REGION Network 97: CLOSED LOW PRESSURE OUTPUT COMMAND MISSING ALARM
   RUNG wire#powerrail
      Contact( #M_VERIFY_LOW_PRESSURE )
      I_Contact( #CYL.CLOSE_LOW_PRESSURE )
      Contact( #CHECK_CLOSED_LOW_PRESSURE_CNC_PLC_SIGNAL )
      wire#w1
      Contact( #O_BYTE_0.CLOSED_LOW_PRESSURE_INPUT )
      Coil( #ALARMS.CLOSED_LOW_PRESSURE_OUTPUT_COMMAND_MISSING_ALARM )
   END_RUNG
   RUNG wire#powerrail
      Contact( #ALARMS.CLOSED_LOW_PRESSURE_OUTPUT_COMMAND_MISSING_ALARM )
      I_Contact( "DB2120_MPP_ITC_IPC".RESET_FAULTS )
   END_RUNG wire#w1
   // the same network as SCL:
   #ALARMS.CLOSED_LOW_PRESSURE_OUTPUT_COMMAND_MISSING_ALARM := ((#M_VERIFY_LOW_PRESSURE AND NOT #CYL.CLOSE_LOW_PRESSURE AND #CHECK_CLOSED_LOW_PRESSURE_CNC_PLC_SIGNAL) OR (#ALARMS.CLOSED_LOW_PRESSURE_OUTPUT_COMMAND_MISSING_ALARM AND NOT "DB2120_MPP_ITC_IPC".RESET_FAULTS)) AND #O_BYTE_0.CLOSED_LOW_PRESSURE_INPUT;
END_REGION

REGION Network 98: OPEN LOW PRESSURE TIME EXCEEDED ALARM
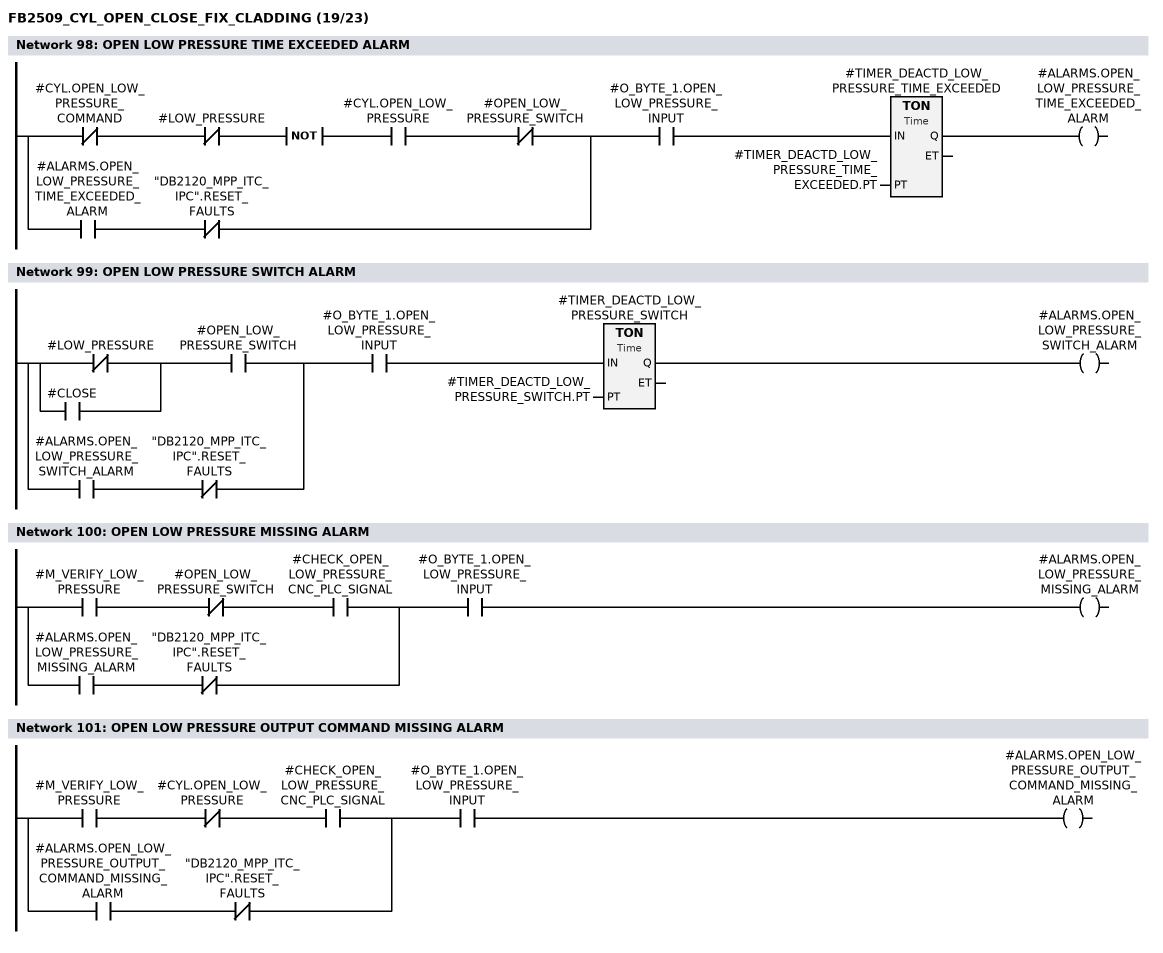
   RUNG wire#powerrail
      I_Contact( #CYL.OPEN_LOW_PRESSURE_COMMAND )
      I_Contact( #LOW_PRESSURE )
      Not()
      Contact( #CYL.OPEN_LOW_PRESSURE )
      I_Contact( #OPEN_LOW_PRESSURE_SWITCH )
      wire#w1
      Contact( #O_BYTE_1.OPEN_LOW_PRESSURE_INPUT )
      { S7_Templates := "time_type := Time" } #TIMER_DEACTD_LOW_PRESSURE_TIME_EXCEEDED.TON(pt := #TIMER_DEACTD_LOW_PRESSURE_TIME_EXCEEDED.PT, et =>)
      Coil( #ALARMS.OPEN_LOW_PRESSURE_TIME_EXCEEDED_ALARM )
   END_RUNG
   RUNG wire#powerrail
      Contact( #ALARMS.OPEN_LOW_PRESSURE_TIME_EXCEEDED_ALARM )
      I_Contact( "DB2120_MPP_ITC_IPC".RESET_FAULTS )
   END_RUNG wire#w1
   // the same network as SCL:
   #TIMER_DEACTD_LOW_PRESSURE_TIME_EXCEEDED(IN := ((NOT (NOT #CYL.OPEN_LOW_PRESSURE_COMMAND AND NOT #LOW_PRESSURE) AND #CYL.OPEN_LOW_PRESSURE AND NOT #OPEN_LOW_PRESSURE_SWITCH) OR (#ALARMS.OPEN_LOW_PRESSURE_TIME_EXCEEDED_ALARM AND NOT "DB2120_MPP_ITC_IPC".RESET_FAULTS)) AND #O_BYTE_1.OPEN_LOW_PRESSURE_INPUT,   // TON
                           PT := #TIMER_DEACTD_LOW_PRESSURE_TIME_EXCEEDED.PT);
   #ALARMS.OPEN_LOW_PRESSURE_TIME_EXCEEDED_ALARM := #TIMER_DEACTD_LOW_PRESSURE_TIME_EXCEEDED.Q;
END_REGION

REGION Network 99: OPEN LOW PRESSURE SWITCH ALARM
   RUNG wire#powerrail
      I_Contact( #LOW_PRESSURE )
      wire#w1
      Contact( #OPEN_LOW_PRESSURE_SWITCH )
      wire#w2
      Contact( #O_BYTE_1.OPEN_LOW_PRESSURE_INPUT )
      { S7_Templates := "time_type := Time" } #TIMER_DEACTD_LOW_PRESSURE_SWITCH.TON(pt := #TIMER_DEACTD_LOW_PRESSURE_SWITCH.PT, et =>)
      Coil( #ALARMS.OPEN_LOW_PRESSURE_SWITCH_ALARM )
   END_RUNG
   RUNG wire#powerrail
      Contact( #CLOSE )
   END_RUNG wire#w1
   RUNG wire#powerrail
      Contact( #ALARMS.OPEN_LOW_PRESSURE_SWITCH_ALARM )
      I_Contact( "DB2120_MPP_ITC_IPC".RESET_FAULTS )
   END_RUNG wire#w2
   // the same network as SCL:
   #TIMER_DEACTD_LOW_PRESSURE_SWITCH(IN := (((NOT #LOW_PRESSURE OR #CLOSE) AND #OPEN_LOW_PRESSURE_SWITCH) OR (#ALARMS.OPEN_LOW_PRESSURE_SWITCH_ALARM AND NOT "DB2120_MPP_ITC_IPC".RESET_FAULTS)) AND #O_BYTE_1.OPEN_LOW_PRESSURE_INPUT,   // TON
                           PT := #TIMER_DEACTD_LOW_PRESSURE_SWITCH.PT);
   #ALARMS.OPEN_LOW_PRESSURE_SWITCH_ALARM := #TIMER_DEACTD_LOW_PRESSURE_SWITCH.Q;
END_REGION

REGION Network 100: OPEN LOW PRESSURE MISSING ALARM
   RUNG wire#powerrail
      Contact( #M_VERIFY_LOW_PRESSURE )
      I_Contact( #OPEN_LOW_PRESSURE_SWITCH )
      Contact( #CHECK_OPEN_LOW_PRESSURE_CNC_PLC_SIGNAL )
      wire#w1
      Contact( #O_BYTE_1.OPEN_LOW_PRESSURE_INPUT )
      Coil( #ALARMS.OPEN_LOW_PRESSURE_MISSING_ALARM )
   END_RUNG
   RUNG wire#powerrail
      Contact( #ALARMS.OPEN_LOW_PRESSURE_MISSING_ALARM )
      I_Contact( "DB2120_MPP_ITC_IPC".RESET_FAULTS )
   END_RUNG wire#w1
   // the same network as SCL:
   #ALARMS.OPEN_LOW_PRESSURE_MISSING_ALARM := ((#M_VERIFY_LOW_PRESSURE AND NOT #OPEN_LOW_PRESSURE_SWITCH AND #CHECK_OPEN_LOW_PRESSURE_CNC_PLC_SIGNAL) OR (#ALARMS.OPEN_LOW_PRESSURE_MISSING_ALARM AND NOT "DB2120_MPP_ITC_IPC".RESET_FAULTS)) AND #O_BYTE_1.OPEN_LOW_PRESSURE_INPUT;
END_REGION

REGION Network 101: OPEN LOW PRESSURE OUTPUT COMMAND MISSING ALARM
   RUNG wire#powerrail
      Contact( #M_VERIFY_LOW_PRESSURE )
      I_Contact( #CYL.OPEN_LOW_PRESSURE )
      Contact( #CHECK_OPEN_LOW_PRESSURE_CNC_PLC_SIGNAL )
      wire#w1
      Contact( #O_BYTE_1.OPEN_LOW_PRESSURE_INPUT )
      Coil( #ALARMS.OPEN_LOW_PRESSURE_OUTPUT_COMMAND_MISSING_ALARM )
   END_RUNG
   RUNG wire#powerrail
      Contact( #ALARMS.OPEN_LOW_PRESSURE_OUTPUT_COMMAND_MISSING_ALARM )
      I_Contact( "DB2120_MPP_ITC_IPC".RESET_FAULTS )
   END_RUNG wire#w1
   // the same network as SCL:
   #ALARMS.OPEN_LOW_PRESSURE_OUTPUT_COMMAND_MISSING_ALARM := ((#M_VERIFY_LOW_PRESSURE AND NOT #CYL.OPEN_LOW_PRESSURE AND #CHECK_OPEN_LOW_PRESSURE_CNC_PLC_SIGNAL) OR (#ALARMS.OPEN_LOW_PRESSURE_OUTPUT_COMMAND_MISSING_ALARM AND NOT "DB2120_MPP_ITC_IPC".RESET_FAULTS)) AND #O_BYTE_1.OPEN_LOW_PRESSURE_INPUT;
END_REGION

REGION Network 102: RETURN HOME POSITION AND STOP END OF CYCLE ALARMS
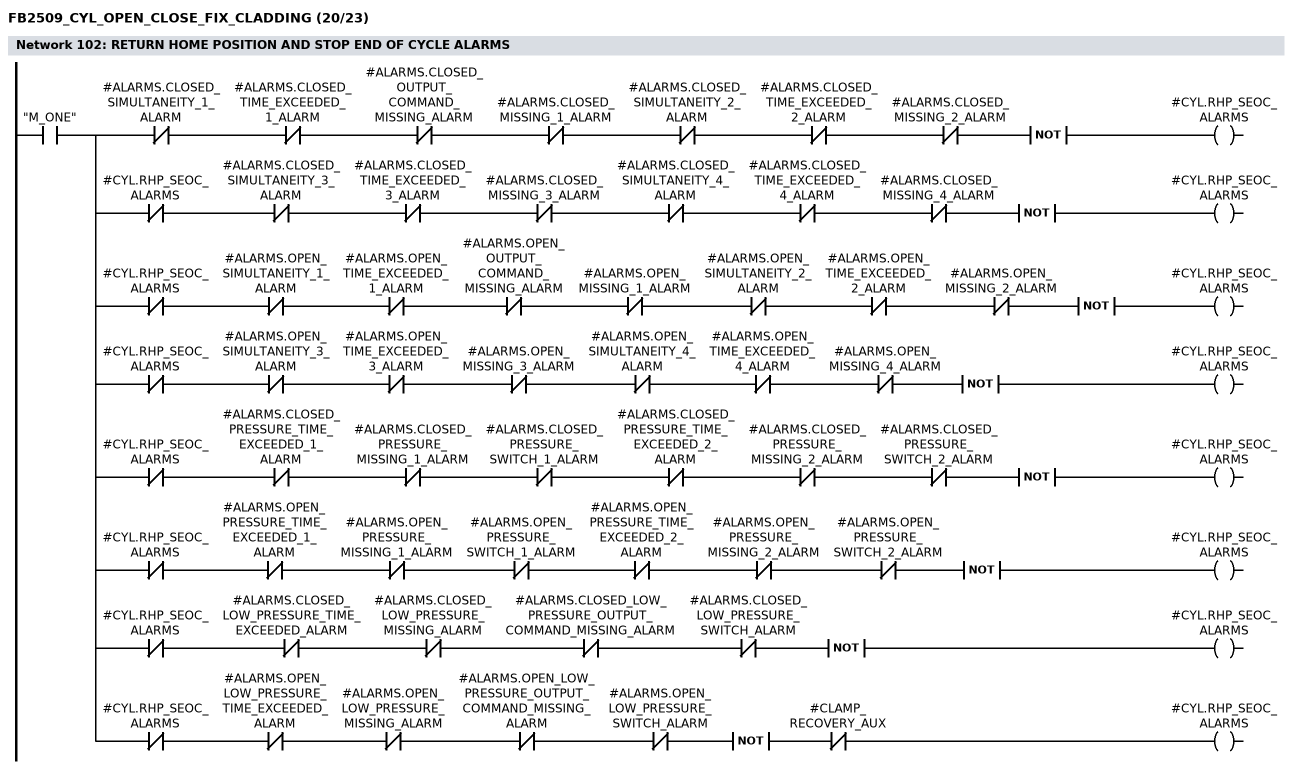
   RUNG wire#powerrail
      Contact( "M_ONE" )
      wire#w1
      I_Contact( #ALARMS.CLOSED_SIMULTANEITY_1_ALARM )
      I_Contact( #ALARMS.CLOSED_TIME_EXCEEDED_1_ALARM )
      I_Contact( #ALARMS.CLOSED_OUTPUT_COMMAND_MISSING_ALARM )
      I_Contact( #ALARMS.CLOSED_MISSING_1_ALARM )
      I_Contact( #ALARMS.CLOSED_SIMULTANEITY_2_ALARM )
      I_Contact( #ALARMS.CLOSED_TIME_EXCEEDED_2_ALARM )
      I_Contact( #ALARMS.CLOSED_MISSING_2_ALARM )
      Not()
      Coil( #CYL.RHP_SEOC_ALARMS )
   END_RUNG
   RUNG wire#w1
      I_Contact( #CYL.RHP_SEOC_ALARMS )
      I_Contact( #ALARMS.CLOSED_SIMULTANEITY_3_ALARM )
      I_Contact( #ALARMS.CLOSED_TIME_EXCEEDED_3_ALARM )
      I_Contact( #ALARMS.CLOSED_MISSING_3_ALARM )
      I_Contact( #ALARMS.CLOSED_SIMULTANEITY_4_ALARM )
      I_Contact( #ALARMS.CLOSED_TIME_EXCEEDED_4_ALARM )
      I_Contact( #ALARMS.CLOSED_MISSING_4_ALARM )
      Not()
      Coil( #CYL.RHP_SEOC_ALARMS )
   END_RUNG
   RUNG wire#w1
      I_Contact( #CYL.RHP_SEOC_ALARMS )
      I_Contact( #ALARMS.OPEN_SIMULTANEITY_1_ALARM )
      I_Contact( #ALARMS.OPEN_TIME_EXCEEDED_1_ALARM )
      I_Contact( #ALARMS.OPEN_OUTPUT_COMMAND_MISSING_ALARM )
      I_Contact( #ALARMS.OPEN_MISSING_1_ALARM )
      I_Contact( #ALARMS.OPEN_SIMULTANEITY_2_ALARM )
      I_Contact( #ALARMS.OPEN_TIME_EXCEEDED_2_ALARM )
      I_Contact( #ALARMS.OPEN_MISSING_2_ALARM )
      Not()
      Coil( #CYL.RHP_SEOC_ALARMS )
   END_RUNG
   RUNG wire#w1
      I_Contact( #CYL.RHP_SEOC_ALARMS )
      I_Contact( #ALARMS.OPEN_SIMULTANEITY_3_ALARM )
      I_Contact( #ALARMS.OPEN_TIME_EXCEEDED_3_ALARM )
      I_Contact( #ALARMS.OPEN_MISSING_3_ALARM )
      I_Contact( #ALARMS.OPEN_SIMULTANEITY_4_ALARM )
      I_Contact( #ALARMS.OPEN_TIME_EXCEEDED_4_ALARM )
      I_Contact( #ALARMS.OPEN_MISSING_4_ALARM )
      Not()
      Coil( #CYL.RHP_SEOC_ALARMS )
   END_RUNG
   RUNG wire#w1
      I_Contact( #CYL.RHP_SEOC_ALARMS )
      I_Contact( #ALARMS.CLOSED_PRESSURE_TIME_EXCEEDED_1_ALARM )
      I_Contact( #ALARMS.CLOSED_PRESSURE_MISSING_1_ALARM )
      I_Contact( #ALARMS.CLOSED_PRESSURE_SWITCH_1_ALARM )
      I_Contact( #ALARMS.CLOSED_PRESSURE_TIME_EXCEEDED_2_ALARM )
      I_Contact( #ALARMS.CLOSED_PRESSURE_MISSING_2_ALARM )
      I_Contact( #ALARMS.CLOSED_PRESSURE_SWITCH_2_ALARM )
      Not()
      Coil( #CYL.RHP_SEOC_ALARMS )
   END_RUNG
   RUNG wire#w1
      I_Contact( #CYL.RHP_SEOC_ALARMS )
      I_Contact( #ALARMS.OPEN_PRESSURE_TIME_EXCEEDED_1_ALARM )
      I_Contact( #ALARMS.OPEN_PRESSURE_MISSING_1_ALARM )
      I_Contact( #ALARMS.OPEN_PRESSURE_SWITCH_1_ALARM )
      I_Contact( #ALARMS.OPEN_PRESSURE_TIME_EXCEEDED_2_ALARM )
      I_Contact( #ALARMS.OPEN_PRESSURE_MISSING_2_ALARM )
      I_Contact( #ALARMS.OPEN_PRESSURE_SWITCH_2_ALARM )
      Not()
      Coil( #CYL.RHP_SEOC_ALARMS )
   END_RUNG
   RUNG wire#w1
      I_Contact( #CYL.RHP_SEOC_ALARMS )
      I_Contact( #ALARMS.CLOSED_LOW_PRESSURE_TIME_EXCEEDED_ALARM )
      I_Contact( #ALARMS.CLOSED_LOW_PRESSURE_MISSING_ALARM )
      I_Contact( #ALARMS.CLOSED_LOW_PRESSURE_OUTPUT_COMMAND_MISSING_ALARM )
      I_Contact( #ALARMS.CLOSED_LOW_PRESSURE_SWITCH_ALARM )
      Not()
      Coil( #CYL.RHP_SEOC_ALARMS )
   END_RUNG
   RUNG wire#w1
      I_Contact( #CYL.RHP_SEOC_ALARMS )
      I_Contact( #ALARMS.OPEN_LOW_PRESSURE_TIME_EXCEEDED_ALARM )
      I_Contact( #ALARMS.OPEN_LOW_PRESSURE_MISSING_ALARM )
      I_Contact( #ALARMS.OPEN_LOW_PRESSURE_OUTPUT_COMMAND_MISSING_ALARM )
      I_Contact( #ALARMS.OPEN_LOW_PRESSURE_SWITCH_ALARM )
      Not()
      I_Contact( #CLAMP_RECOVERY_AUX )
      Coil( #CYL.RHP_SEOC_ALARMS )
   END_RUNG
   // the same network as SCL:
   #CYL.RHP_SEOC_ALARMS := NOT ("M_ONE" AND NOT #ALARMS.CLOSED_SIMULTANEITY_1_ALARM AND NOT #ALARMS.CLOSED_TIME_EXCEEDED_1_ALARM AND NOT #ALARMS.CLOSED_OUTPUT_COMMAND_MISSING_ALARM AND NOT #ALARMS.CLOSED_MISSING_1_ALARM AND NOT #ALARMS.CLOSED_SIMULTANEITY_2_ALARM AND NOT #ALARMS.CLOSED_TIME_EXCEEDED_2_ALARM AND NOT #ALARMS.CLOSED_MISSING_2_ALARM);
   #CYL.RHP_SEOC_ALARMS := NOT ("M_ONE" AND NOT #CYL.RHP_SEOC_ALARMS AND NOT #ALARMS.CLOSED_SIMULTANEITY_3_ALARM AND NOT #ALARMS.CLOSED_TIME_EXCEEDED_3_ALARM AND NOT #ALARMS.CLOSED_MISSING_3_ALARM AND NOT #ALARMS.CLOSED_SIMULTANEITY_4_ALARM AND NOT #ALARMS.CLOSED_TIME_EXCEEDED_4_ALARM AND NOT #ALARMS.CLOSED_MISSING_4_ALARM);
   #CYL.RHP_SEOC_ALARMS := NOT ("M_ONE" AND NOT #CYL.RHP_SEOC_ALARMS AND NOT #ALARMS.OPEN_SIMULTANEITY_1_ALARM AND NOT #ALARMS.OPEN_TIME_EXCEEDED_1_ALARM AND NOT #ALARMS.OPEN_OUTPUT_COMMAND_MISSING_ALARM AND NOT #ALARMS.OPEN_MISSING_1_ALARM AND NOT #ALARMS.OPEN_SIMULTANEITY_2_ALARM AND NOT #ALARMS.OPEN_TIME_EXCEEDED_2_ALARM AND NOT #ALARMS.OPEN_MISSING_2_ALARM);
   #CYL.RHP_SEOC_ALARMS := NOT ("M_ONE" AND NOT #CYL.RHP_SEOC_ALARMS AND NOT #ALARMS.OPEN_SIMULTANEITY_3_ALARM AND NOT #ALARMS.OPEN_TIME_EXCEEDED_3_ALARM AND NOT #ALARMS.OPEN_MISSING_3_ALARM AND NOT #ALARMS.OPEN_SIMULTANEITY_4_ALARM AND NOT #ALARMS.OPEN_TIME_EXCEEDED_4_ALARM AND NOT #ALARMS.OPEN_MISSING_4_ALARM);
   #CYL.RHP_SEOC_ALARMS := NOT ("M_ONE" AND NOT #CYL.RHP_SEOC_ALARMS AND NOT #ALARMS.CLOSED_PRESSURE_TIME_EXCEEDED_1_ALARM AND NOT #ALARMS.CLOSED_PRESSURE_MISSING_1_ALARM AND NOT #ALARMS.CLOSED_PRESSURE_SWITCH_1_ALARM AND NOT #ALARMS.CLOSED_PRESSURE_TIME_EXCEEDED_2_ALARM AND NOT #ALARMS.CLOSED_PRESSURE_MISSING_2_ALARM AND NOT #ALARMS.CLOSED_PRESSURE_SWITCH_2_ALARM);
   #CYL.RHP_SEOC_ALARMS := NOT ("M_ONE" AND NOT #CYL.RHP_SEOC_ALARMS AND NOT #ALARMS.OPEN_PRESSURE_TIME_EXCEEDED_1_ALARM AND NOT #ALARMS.OPEN_PRESSURE_MISSING_1_ALARM AND NOT #ALARMS.OPEN_PRESSURE_SWITCH_1_ALARM AND NOT #ALARMS.OPEN_PRESSURE_TIME_EXCEEDED_2_ALARM AND NOT #ALARMS.OPEN_PRESSURE_MISSING_2_ALARM AND NOT #ALARMS.OPEN_PRESSURE_SWITCH_2_ALARM);
   #CYL.RHP_SEOC_ALARMS := NOT ("M_ONE" AND NOT #CYL.RHP_SEOC_ALARMS AND NOT #ALARMS.CLOSED_LOW_PRESSURE_TIME_EXCEEDED_ALARM AND NOT #ALARMS.CLOSED_LOW_PRESSURE_MISSING_ALARM AND NOT #ALARMS.CLOSED_LOW_PRESSURE_OUTPUT_COMMAND_MISSING_ALARM AND NOT #ALARMS.CLOSED_LOW_PRESSURE_SWITCH_ALARM);
   #CYL.RHP_SEOC_ALARMS := NOT ("M_ONE" AND NOT #CYL.RHP_SEOC_ALARMS AND NOT #ALARMS.OPEN_LOW_PRESSURE_TIME_EXCEEDED_ALARM AND NOT #ALARMS.OPEN_LOW_PRESSURE_MISSING_ALARM AND NOT #ALARMS.OPEN_LOW_PRESSURE_OUTPUT_COMMAND_MISSING_ALARM AND NOT #ALARMS.OPEN_LOW_PRESSURE_SWITCH_ALARM) AND NOT #CLAMP_RECOVERY_AUX;
END_REGION

REGION Network 103: RETURN HOME POSITION AND STOP END OF CYCLE ALARMS
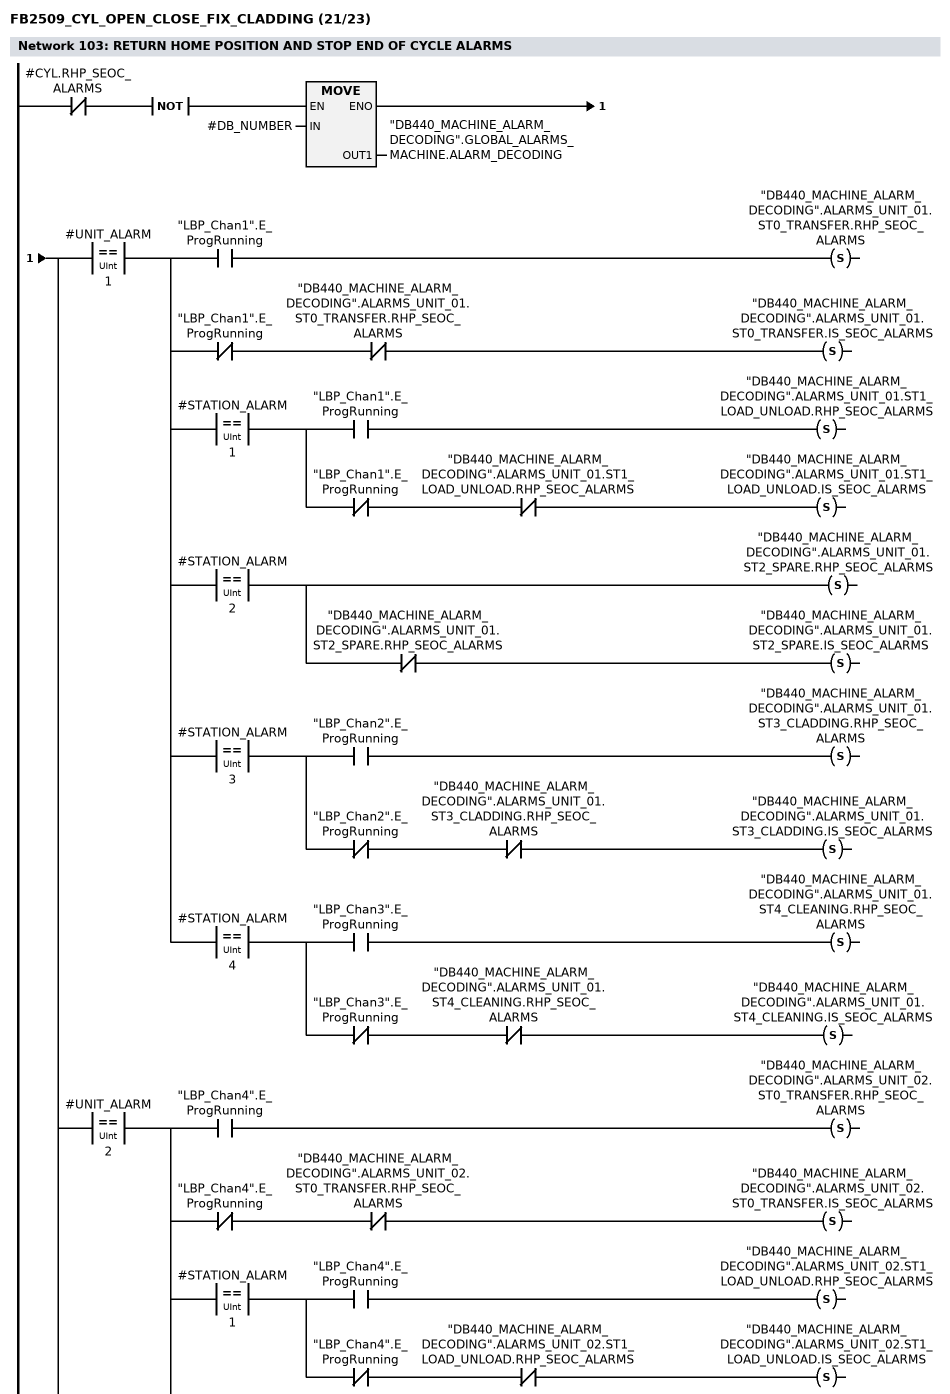
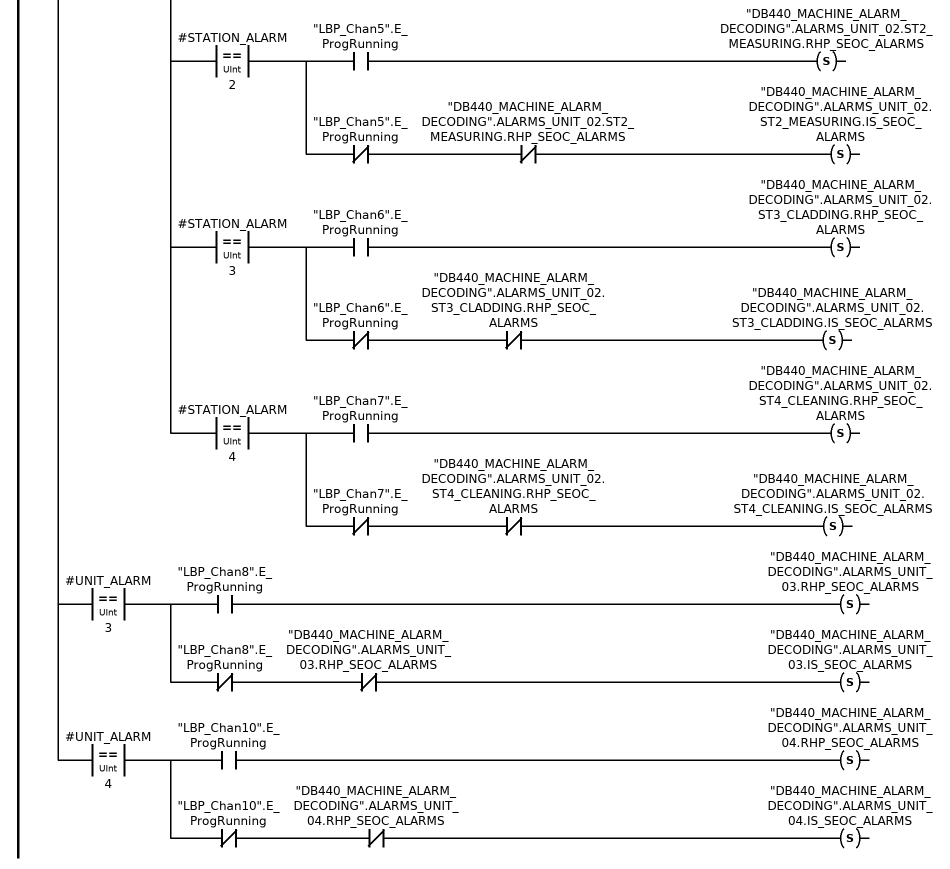
   RUNG wire#powerrail
      I_Contact( #CYL.RHP_SEOC_ALARMS )
      Not()
      { S7_GenerateENO := "TRUE" } Move(in := #DB_NUMBER, out1 => "DB440_MACHINE_ALARM_DECODING".GLOBAL_ALARMS_MACHINE.ALARM_DECODING)
      wire#w1
      { S7_Templates := "SrcType := UInt" } EQ_Contact(in1 := #UNIT_ALARM, in2 := 1)
      wire#w2
      Contact( "LBP_Chan1".E_ProgRunning )
      S_Coil( "DB440_MACHINE_ALARM_DECODING".ALARMS_UNIT_01.ST0_TRANSFER.RHP_SEOC_ALARMS )
   END_RUNG
   RUNG wire#w2
      I_Contact( "LBP_Chan1".E_ProgRunning )
      I_Contact( "DB440_MACHINE_ALARM_DECODING".ALARMS_UNIT_01.ST0_TRANSFER.RHP_SEOC_ALARMS )
      S_Coil( "DB440_MACHINE_ALARM_DECODING".ALARMS_UNIT_01.ST0_TRANSFER.IS_SEOC_ALARMS )
   END_RUNG
   RUNG wire#w2
      { S7_Templates := "SrcType := UInt" } EQ_Contact(in1 := #STATION_ALARM, in2 := 1)
      wire#w3
      Contact( "LBP_Chan1".E_ProgRunning )
      S_Coil( "DB440_MACHINE_ALARM_DECODING".ALARMS_UNIT_01.ST1_LOAD_UNLOAD.RHP_SEOC_ALARMS )
   END_RUNG
   RUNG wire#w3
      I_Contact( "LBP_Chan1".E_ProgRunning )
      I_Contact( "DB440_MACHINE_ALARM_DECODING".ALARMS_UNIT_01.ST1_LOAD_UNLOAD.RHP_SEOC_ALARMS )
      S_Coil( "DB440_MACHINE_ALARM_DECODING".ALARMS_UNIT_01.ST1_LOAD_UNLOAD.IS_SEOC_ALARMS )
   END_RUNG
   RUNG wire#w2
      { S7_Templates := "SrcType := UInt" } EQ_Contact(in1 := #STATION_ALARM, in2 := 2)
      wire#w4
      S_Coil( "DB440_MACHINE_ALARM_DECODING".ALARMS_UNIT_01.ST2_SPARE.RHP_SEOC_ALARMS )
   END_RUNG
   RUNG wire#w4
      I_Contact( "DB440_MACHINE_ALARM_DECODING".ALARMS_UNIT_01.ST2_SPARE.RHP_SEOC_ALARMS )
      S_Coil( "DB440_MACHINE_ALARM_DECODING".ALARMS_UNIT_01.ST2_SPARE.IS_SEOC_ALARMS )
   END_RUNG
   RUNG wire#w2
      { S7_Templates := "SrcType := UInt" } EQ_Contact(in1 := #STATION_ALARM, in2 := 3)
      wire#w5
      Contact( "LBP_Chan2".E_ProgRunning )
      S_Coil( "DB440_MACHINE_ALARM_DECODING".ALARMS_UNIT_01.ST3_CLADDING.RHP_SEOC_ALARMS )
   END_RUNG
   RUNG wire#w5
      I_Contact( "LBP_Chan2".E_ProgRunning )
      I_Contact( "DB440_MACHINE_ALARM_DECODING".ALARMS_UNIT_01.ST3_CLADDING.RHP_SEOC_ALARMS )
      S_Coil( "DB440_MACHINE_ALARM_DECODING".ALARMS_UNIT_01.ST3_CLADDING.IS_SEOC_ALARMS )
   END_RUNG
   RUNG wire#w2
      { S7_Templates := "SrcType := UInt" } EQ_Contact(in1 := #STATION_ALARM, in2 := 4)
      wire#w6
      Contact( "LBP_Chan3".E_ProgRunning )
      S_Coil( "DB440_MACHINE_ALARM_DECODING".ALARMS_UNIT_01.ST4_CLEANING.RHP_SEOC_ALARMS )
   END_RUNG
   RUNG wire#w6
      I_Contact( "LBP_Chan3".E_ProgRunning )
      I_Contact( "DB440_MACHINE_ALARM_DECODING".ALARMS_UNIT_01.ST4_CLEANING.RHP_SEOC_ALARMS )
      S_Coil( "DB440_MACHINE_ALARM_DECODING".ALARMS_UNIT_01.ST4_CLEANING.IS_SEOC_ALARMS )
   END_RUNG
   RUNG wire#w1
      { S7_Templates := "SrcType := UInt" } EQ_Contact(in1 := #UNIT_ALARM, in2 := 2)
      wire#w7
      Contact( "LBP_Chan4".E_ProgRunning )
      S_Coil( "DB440_MACHINE_ALARM_DECODING".ALARMS_UNIT_02.ST0_TRANSFER.RHP_SEOC_ALARMS )
   END_RUNG
   RUNG wire#w7
      I_Contact( "LBP_Chan4".E_ProgRunning )
      I_Contact( "DB440_MACHINE_ALARM_DECODING".ALARMS_UNIT_02.ST0_TRANSFER.RHP_SEOC_ALARMS )
      S_Coil( "DB440_MACHINE_ALARM_DECODING".ALARMS_UNIT_02.ST0_TRANSFER.IS_SEOC_ALARMS )
   END_RUNG
   RUNG wire#w7
      { S7_Templates := "SrcType := UInt" } EQ_Contact(in1 := #STATION_ALARM, in2 := 1)
      wire#w8
      Contact( "LBP_Chan4".E_ProgRunning )
      S_Coil( "DB440_MACHINE_ALARM_DECODING".ALARMS_UNIT_02.ST1_LOAD_UNLOAD.RHP_SEOC_ALARMS )
   END_RUNG
   RUNG wire#w8
      I_Contact( "LBP_Chan4".E_ProgRunning )
      I_Contact( "DB440_MACHINE_ALARM_DECODING".ALARMS_UNIT_02.ST1_LOAD_UNLOAD.RHP_SEOC_ALARMS )
      S_Coil( "DB440_MACHINE_ALARM_DECODING".ALARMS_UNIT_02.ST1_LOAD_UNLOAD.IS_SEOC_ALARMS )
   END_RUNG
   RUNG wire#w7
      { S7_Templates := "SrcType := UInt" } EQ_Contact(in1 := #STATION_ALARM, in2 := 2)
      wire#w9
      Contact( "LBP_Chan5".E_ProgRunning )
      S_Coil( "DB440_MACHINE_ALARM_DECODING".ALARMS_UNIT_02.ST2_MEASURING.RHP_SEOC_ALARMS )
   END_RUNG
   RUNG wire#w9
      I_Contact( "LBP_Chan5".E_ProgRunning )
      I_Contact( "DB440_MACHINE_ALARM_DECODING".ALARMS_UNIT_02.ST2_MEASURING.RHP_SEOC_ALARMS )
      S_Coil( "DB440_MACHINE_ALARM_DECODING".ALARMS_UNIT_02.ST2_MEASURING.IS_SEOC_ALARMS )
   END_RUNG
   RUNG wire#w7
      { S7_Templates := "SrcType := UInt" } EQ_Contact(in1 := #STATION_ALARM, in2 := 3)
      wire#w10
      Contact( "LBP_Chan6".E_ProgRunning )
      S_Coil( "DB440_MACHINE_ALARM_DECODING".ALARMS_UNIT_02.ST3_CLADDING.RHP_SEOC_ALARMS )
   END_RUNG
   RUNG wire#w10
      I_Contact( "LBP_Chan6".E_ProgRunning )
      I_Contact( "DB440_MACHINE_ALARM_DECODING".ALARMS_UNIT_02.ST3_CLADDING.RHP_SEOC_ALARMS )
      S_Coil( "DB440_MACHINE_ALARM_DECODING".ALARMS_UNIT_02.ST3_CLADDING.IS_SEOC_ALARMS )
   END_RUNG
   RUNG wire#w7
      { S7_Templates := "SrcType := UInt" } EQ_Contact(in1 := #STATION_ALARM, in2 := 4)
      wire#w11
      Contact( "LBP_Chan7".E_ProgRunning )
      S_Coil( "DB440_MACHINE_ALARM_DECODING".ALARMS_UNIT_02.ST4_CLEANING.RHP_SEOC_ALARMS )
   END_RUNG
   RUNG wire#w11
      I_Contact( "LBP_Chan7".E_ProgRunning )
      I_Contact( "DB440_MACHINE_ALARM_DECODING".ALARMS_UNIT_02.ST4_CLEANING.RHP_SEOC_ALARMS )
      S_Coil( "DB440_MACHINE_ALARM_DECODING".ALARMS_UNIT_02.ST4_CLEANING.IS_SEOC_ALARMS )
   END_RUNG
   RUNG wire#w1
      { S7_Templates := "SrcType := UInt" } EQ_Contact(in1 := #UNIT_ALARM, in2 := 3)
      wire#w12
      Contact( "LBP_Chan8".E_ProgRunning )
      S_Coil( "DB440_MACHINE_ALARM_DECODING".ALARMS_UNIT_03.RHP_SEOC_ALARMS )
   END_RUNG
   RUNG wire#w12
      I_Contact( "LBP_Chan8".E_ProgRunning )
      I_Contact( "DB440_MACHINE_ALARM_DECODING".ALARMS_UNIT_03.RHP_SEOC_ALARMS )
      S_Coil( "DB440_MACHINE_ALARM_DECODING".ALARMS_UNIT_03.IS_SEOC_ALARMS )
   END_RUNG
   RUNG wire#w1
      { S7_Templates := "SrcType := UInt" } EQ_Contact(in1 := #UNIT_ALARM, in2 := 4)
      wire#w13
      Contact( "LBP_Chan10".E_ProgRunning )
      S_Coil( "DB440_MACHINE_ALARM_DECODING".ALARMS_UNIT_04.RHP_SEOC_ALARMS )
   END_RUNG
   RUNG wire#w13
      I_Contact( "LBP_Chan10".E_ProgRunning )
      I_Contact( "DB440_MACHINE_ALARM_DECODING".ALARMS_UNIT_04.RHP_SEOC_ALARMS )
      S_Coil( "DB440_MACHINE_ALARM_DECODING".ALARMS_UNIT_04.IS_SEOC_ALARMS )
   END_RUNG
   // the same network as SCL:
   // ENO of a box is taken as its EN; it also drops when the box reports an error
   #_w1 := NOT (NOT #CYL.RHP_SEOC_ALARMS);
   IF #_w1 THEN "DB440_MACHINE_ALARM_DECODING".GLOBAL_ALARMS_MACHINE.ALARM_DECODING := #DB_NUMBER; END_IF;
   #_w2 := #_w1 AND (#UNIT_ALARM = 1);
   IF #_w2 AND "LBP_Chan1".E_ProgRunning THEN
       "DB440_MACHINE_ALARM_DECODING".ALARMS_UNIT_01.ST0_TRANSFER.RHP_SEOC_ALARMS := TRUE;
   END_IF;
   IF #_w2 AND NOT "LBP_Chan1".E_ProgRunning AND NOT "DB440_MACHINE_ALARM_DECODING".ALARMS_UNIT_01.ST0_TRANSFER.RHP_SEOC_ALARMS THEN
       "DB440_MACHINE_ALARM_DECODING".ALARMS_UNIT_01.ST0_TRANSFER.IS_SEOC_ALARMS := TRUE;
   END_IF;
   #_w3 := #_w2 AND (#STATION_ALARM = 1);
   IF #_w3 AND "LBP_Chan1".E_ProgRunning THEN
       "DB440_MACHINE_ALARM_DECODING".ALARMS_UNIT_01.ST1_LOAD_UNLOAD.RHP_SEOC_ALARMS := TRUE;
   END_IF;
   IF #_w3 AND NOT "LBP_Chan1".E_ProgRunning AND NOT "DB440_MACHINE_ALARM_DECODING".ALARMS_UNIT_01.ST1_LOAD_UNLOAD.RHP_SEOC_ALARMS THEN
       "DB440_MACHINE_ALARM_DECODING".ALARMS_UNIT_01.ST1_LOAD_UNLOAD.IS_SEOC_ALARMS := TRUE;
   END_IF;
   #_w4 := #_w2 AND (#STATION_ALARM = 2);
   IF #_w4 THEN "DB440_MACHINE_ALARM_DECODING".ALARMS_UNIT_01.ST2_SPARE.RHP_SEOC_ALARMS := TRUE; END_IF;
   IF #_w4 AND NOT "DB440_MACHINE_ALARM_DECODING".ALARMS_UNIT_01.ST2_SPARE.RHP_SEOC_ALARMS THEN
       "DB440_MACHINE_ALARM_DECODING".ALARMS_UNIT_01.ST2_SPARE.IS_SEOC_ALARMS := TRUE;
   END_IF;
   #_w5 := #_w2 AND (#STATION_ALARM = 3);
   IF #_w5 AND "LBP_Chan2".E_ProgRunning THEN
       "DB440_MACHINE_ALARM_DECODING".ALARMS_UNIT_01.ST3_CLADDING.RHP_SEOC_ALARMS := TRUE;
   END_IF;
   IF #_w5 AND NOT "LBP_Chan2".E_ProgRunning AND NOT "DB440_MACHINE_ALARM_DECODING".ALARMS_UNIT_01.ST3_CLADDING.RHP_SEOC_ALARMS THEN
       "DB440_MACHINE_ALARM_DECODING".ALARMS_UNIT_01.ST3_CLADDING.IS_SEOC_ALARMS := TRUE;
   END_IF;
   #_w6 := #_w2 AND (#STATION_ALARM = 4);
   IF #_w6 AND "LBP_Chan3".E_ProgRunning THEN
       "DB440_MACHINE_ALARM_DECODING".ALARMS_UNIT_01.ST4_CLEANING.RHP_SEOC_ALARMS := TRUE;
   END_IF;
   IF #_w6 AND NOT "LBP_Chan3".E_ProgRunning AND NOT "DB440_MACHINE_ALARM_DECODING".ALARMS_UNIT_01.ST4_CLEANING.RHP_SEOC_ALARMS THEN
       "DB440_MACHINE_ALARM_DECODING".ALARMS_UNIT_01.ST4_CLEANING.IS_SEOC_ALARMS := TRUE;
   END_IF;
   #_w7 := #_w1 AND (#UNIT_ALARM = 2);
   IF #_w7 AND "LBP_Chan4".E_ProgRunning THEN
       "DB440_MACHINE_ALARM_DECODING".ALARMS_UNIT_02.ST0_TRANSFER.RHP_SEOC_ALARMS := TRUE;
   END_IF;
   IF #_w7 AND NOT "LBP_Chan4".E_ProgRunning AND NOT "DB440_MACHINE_ALARM_DECODING".ALARMS_UNIT_02.ST0_TRANSFER.RHP_SEOC_ALARMS THEN
       "DB440_MACHINE_ALARM_DECODING".ALARMS_UNIT_02.ST0_TRANSFER.IS_SEOC_ALARMS := TRUE;
   END_IF;
   #_w8 := #_w7 AND (#STATION_ALARM = 1);
   IF #_w8 AND "LBP_Chan4".E_ProgRunning THEN
       "DB440_MACHINE_ALARM_DECODING".ALARMS_UNIT_02.ST1_LOAD_UNLOAD.RHP_SEOC_ALARMS := TRUE;
   END_IF;
   IF #_w8 AND NOT "LBP_Chan4".E_ProgRunning AND NOT "DB440_MACHINE_ALARM_DECODING".ALARMS_UNIT_02.ST1_LOAD_UNLOAD.RHP_SEOC_ALARMS THEN
       "DB440_MACHINE_ALARM_DECODING".ALARMS_UNIT_02.ST1_LOAD_UNLOAD.IS_SEOC_ALARMS := TRUE;
   END_IF;
   #_w9 := #_w7 AND (#STATION_ALARM = 2);
   IF #_w9 AND "LBP_Chan5".E_ProgRunning THEN
       "DB440_MACHINE_ALARM_DECODING".ALARMS_UNIT_02.ST2_MEASURING.RHP_SEOC_ALARMS := TRUE;
   END_IF;
   IF #_w9 AND NOT "LBP_Chan5".E_ProgRunning AND NOT "DB440_MACHINE_ALARM_DECODING".ALARMS_UNIT_02.ST2_MEASURING.RHP_SEOC_ALARMS THEN
       "DB440_MACHINE_ALARM_DECODING".ALARMS_UNIT_02.ST2_MEASURING.IS_SEOC_ALARMS := TRUE;
   END_IF;
   #_w10 := #_w7 AND (#STATION_ALARM = 3);
   IF #_w10 AND "LBP_Chan6".E_ProgRunning THEN
       "DB440_MACHINE_ALARM_DECODING".ALARMS_UNIT_02.ST3_CLADDING.RHP_SEOC_ALARMS := TRUE;
   END_IF;
   IF #_w10 AND NOT "LBP_Chan6".E_ProgRunning AND NOT "DB440_MACHINE_ALARM_DECODING".ALARMS_UNIT_02.ST3_CLADDING.RHP_SEOC_ALARMS THEN
       "DB440_MACHINE_ALARM_DECODING".ALARMS_UNIT_02.ST3_CLADDING.IS_SEOC_ALARMS := TRUE;
   END_IF;
   #_w11 := #_w7 AND (#STATION_ALARM = 4);
   IF #_w11 AND "LBP_Chan7".E_ProgRunning THEN
       "DB440_MACHINE_ALARM_DECODING".ALARMS_UNIT_02.ST4_CLEANING.RHP_SEOC_ALARMS := TRUE;
   END_IF;
   IF #_w11 AND NOT "LBP_Chan7".E_ProgRunning AND NOT "DB440_MACHINE_ALARM_DECODING".ALARMS_UNIT_02.ST4_CLEANING.RHP_SEOC_ALARMS THEN
       "DB440_MACHINE_ALARM_DECODING".ALARMS_UNIT_02.ST4_CLEANING.IS_SEOC_ALARMS := TRUE;
   END_IF;
   #_w12 := #_w1 AND (#UNIT_ALARM = 3);
   IF #_w12 AND "LBP_Chan8".E_ProgRunning THEN
       "DB440_MACHINE_ALARM_DECODING".ALARMS_UNIT_03.RHP_SEOC_ALARMS := TRUE;
   END_IF;
   IF #_w12 AND NOT "LBP_Chan8".E_ProgRunning AND NOT "DB440_MACHINE_ALARM_DECODING".ALARMS_UNIT_03.RHP_SEOC_ALARMS THEN
       "DB440_MACHINE_ALARM_DECODING".ALARMS_UNIT_03.IS_SEOC_ALARMS := TRUE;
   END_IF;
   #_w13 := #_w1 AND (#UNIT_ALARM = 4);
   IF #_w13 AND "LBP_Chan10".E_ProgRunning THEN
       "DB440_MACHINE_ALARM_DECODING".ALARMS_UNIT_04.RHP_SEOC_ALARMS := TRUE;
   END_IF;
   IF #_w13 AND NOT "LBP_Chan10".E_ProgRunning AND NOT "DB440_MACHINE_ALARM_DECODING".ALARMS_UNIT_04.RHP_SEOC_ALARMS THEN
       "DB440_MACHINE_ALARM_DECODING".ALARMS_UNIT_04.IS_SEOC_ALARMS := TRUE;
   END_IF;
END_REGION

REGION Network 104: ANY ACTIVE ALARM
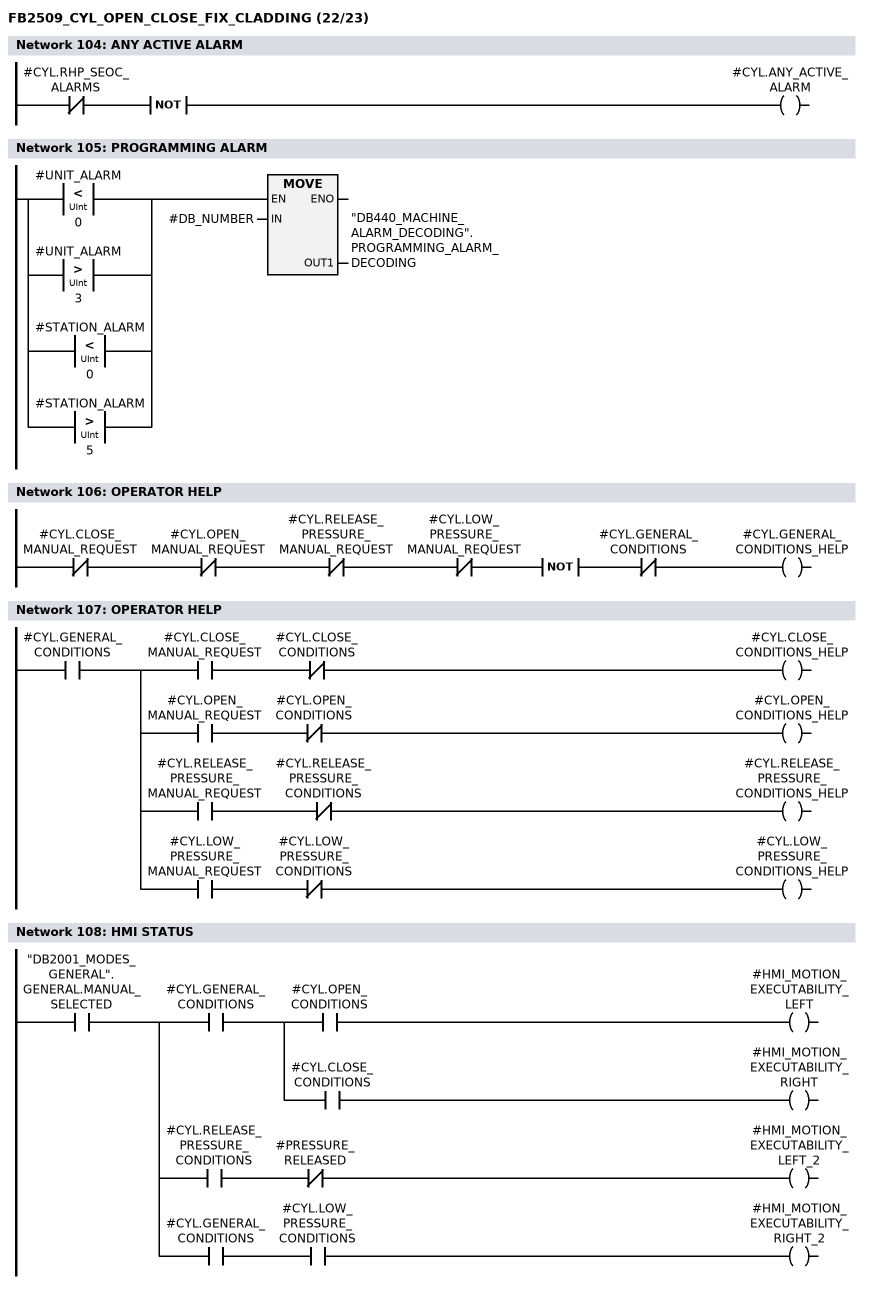
   RUNG wire#powerrail
      I_Contact( #CYL.RHP_SEOC_ALARMS )
      Not()
      Coil( #CYL.ANY_ACTIVE_ALARM )
   END_RUNG
   // the same network as SCL:
   #CYL.ANY_ACTIVE_ALARM := NOT (NOT #CYL.RHP_SEOC_ALARMS);
END_REGION

REGION Network 105: PROGRAMMING ALARM
   RUNG wire#powerrail
      { S7_Templates := "SrcType := UInt" } LT_Contact(in1 := #UNIT_ALARM, in2 := 0)
      wire#w1
      Move(in := #DB_NUMBER, out1 => "DB440_MACHINE_ALARM_DECODING".PROGRAMMING_ALARM_DECODING)
   END_RUNG
   RUNG wire#powerrail
      { S7_Templates := "SrcType := UInt" } GT_Contact(in1 := #UNIT_ALARM, in2 := 3)
   END_RUNG wire#w1
   RUNG wire#powerrail
      { S7_Templates := "SrcType := UInt" } LT_Contact(in1 := #STATION_ALARM, in2 := 0)
   END_RUNG wire#w1
   RUNG wire#powerrail
      { S7_Templates := "SrcType := UInt" } GT_Contact(in1 := #STATION_ALARM, in2 := 5)
   END_RUNG wire#w1
   // the same network as SCL:
   IF (#UNIT_ALARM < 0) OR (#UNIT_ALARM > 3) OR (#STATION_ALARM < 0) OR (#STATION_ALARM > 5) THEN
       "DB440_MACHINE_ALARM_DECODING".PROGRAMMING_ALARM_DECODING := #DB_NUMBER;
   END_IF;
END_REGION

REGION Network 106: OPERATOR HELP
   RUNG wire#powerrail
      I_Contact( #CYL.CLOSE_MANUAL_REQUEST )
      I_Contact( #CYL.OPEN_MANUAL_REQUEST )
      I_Contact( #CYL.RELEASE_PRESSURE_MANUAL_REQUEST )
      I_Contact( #CYL.LOW_PRESSURE_MANUAL_REQUEST )
      Not()
      I_Contact( #CYL.GENERAL_CONDITIONS )
      Coil( #CYL.GENERAL_CONDITIONS_HELP )
   END_RUNG
   // the same network as SCL:
   #CYL.GENERAL_CONDITIONS_HELP := NOT (NOT #CYL.CLOSE_MANUAL_REQUEST AND NOT #CYL.OPEN_MANUAL_REQUEST AND NOT #CYL.RELEASE_PRESSURE_MANUAL_REQUEST AND NOT #CYL.LOW_PRESSURE_MANUAL_REQUEST) AND NOT #CYL.GENERAL_CONDITIONS;
END_REGION

REGION Network 107: OPERATOR HELP
   RUNG wire#powerrail
      Contact( #CYL.GENERAL_CONDITIONS )
      wire#w1
      Contact( #CYL.CLOSE_MANUAL_REQUEST )
      I_Contact( #CYL.CLOSE_CONDITIONS )
      Coil( #CYL.CLOSE_CONDITIONS_HELP )
   END_RUNG
   RUNG wire#w1
      Contact( #CYL.OPEN_MANUAL_REQUEST )
      I_Contact( #CYL.OPEN_CONDITIONS )
      Coil( #CYL.OPEN_CONDITIONS_HELP )
   END_RUNG
   RUNG wire#w1
      Contact( #CYL.RELEASE_PRESSURE_MANUAL_REQUEST )
      I_Contact( #CYL.RELEASE_PRESSURE_CONDITIONS )
      Coil( #CYL.RELEASE_PRESSURE_CONDITIONS_HELP )
   END_RUNG
   RUNG wire#w1
      Contact( #CYL.LOW_PRESSURE_MANUAL_REQUEST )
      I_Contact( #CYL.LOW_PRESSURE_CONDITIONS )
      Coil( #CYL.LOW_PRESSURE_CONDITIONS_HELP )
   END_RUNG
   // the same network as SCL:
   #CYL.CLOSE_CONDITIONS_HELP := #CYL.GENERAL_CONDITIONS AND #CYL.CLOSE_MANUAL_REQUEST AND NOT #CYL.CLOSE_CONDITIONS;
   #CYL.OPEN_CONDITIONS_HELP := #CYL.GENERAL_CONDITIONS AND #CYL.OPEN_MANUAL_REQUEST AND NOT #CYL.OPEN_CONDITIONS;
   #CYL.RELEASE_PRESSURE_CONDITIONS_HELP := #CYL.GENERAL_CONDITIONS AND #CYL.RELEASE_PRESSURE_MANUAL_REQUEST AND NOT #CYL.RELEASE_PRESSURE_CONDITIONS;
   #CYL.LOW_PRESSURE_CONDITIONS_HELP := #CYL.GENERAL_CONDITIONS AND #CYL.LOW_PRESSURE_MANUAL_REQUEST AND NOT #CYL.LOW_PRESSURE_CONDITIONS;
END_REGION

REGION Network 108: HMI STATUS
   RUNG wire#powerrail
      Contact( "DB2001_MODES_GENERAL".GENERAL.MANUAL_SELECTED )
      wire#w1
      Contact( #CYL.GENERAL_CONDITIONS )
      wire#w2
      Contact( #CYL.OPEN_CONDITIONS )
      Coil( #HMI_MOTION_EXECUTABILITY_LEFT )
   END_RUNG
   RUNG wire#w2
      Contact( #CYL.CLOSE_CONDITIONS )
      Coil( #HMI_MOTION_EXECUTABILITY_RIGHT )
   END_RUNG
   RUNG wire#w1
      Contact( #CYL.RELEASE_PRESSURE_CONDITIONS )
      I_Contact( #PRESSURE_RELEASED )
      Coil( #HMI_MOTION_EXECUTABILITY_LEFT_2 )
   END_RUNG
   RUNG wire#w1
      Contact( #CYL.GENERAL_CONDITIONS )
      Contact( #CYL.LOW_PRESSURE_CONDITIONS )
      Coil( #HMI_MOTION_EXECUTABILITY_RIGHT_2 )
   END_RUNG
   // the same network as SCL:
   #_w1 := "DB2001_MODES_GENERAL".GENERAL.MANUAL_SELECTED AND #CYL.GENERAL_CONDITIONS;
   #HMI_MOTION_EXECUTABILITY_LEFT := #_w1 AND #CYL.OPEN_CONDITIONS;
   #HMI_MOTION_EXECUTABILITY_RIGHT := #_w1 AND #CYL.CLOSE_CONDITIONS;
   #HMI_MOTION_EXECUTABILITY_LEFT_2 := "DB2001_MODES_GENERAL".GENERAL.MANUAL_SELECTED AND #CYL.RELEASE_PRESSURE_CONDITIONS AND NOT #PRESSURE_RELEASED;
   #HMI_MOTION_EXECUTABILITY_RIGHT_2 := "DB2001_MODES_GENERAL".GENERAL.MANUAL_SELECTED AND #CYL.GENERAL_CONDITIONS AND #CYL.LOW_PRESSURE_CONDITIONS;
END_REGION

REGION Network 109: HMI STATUS
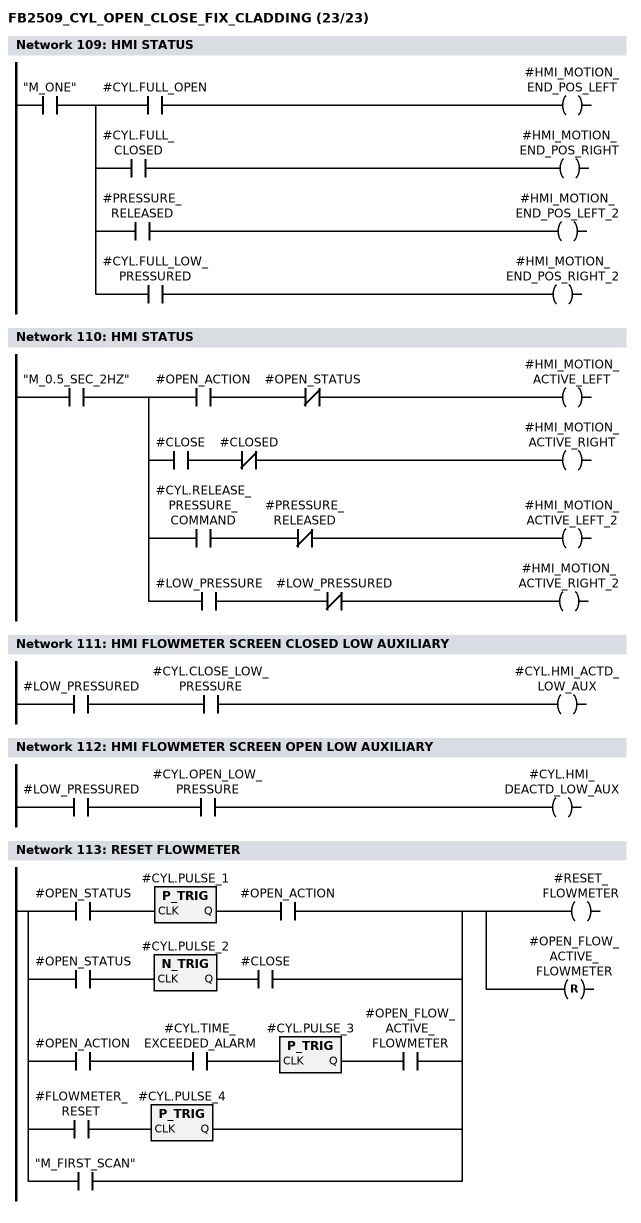
   RUNG wire#powerrail
      Contact( "M_ONE" )
      wire#w1
      Contact( #CYL.FULL_OPEN )
      Coil( #HMI_MOTION_END_POS_LEFT )
   END_RUNG
   RUNG wire#w1
      Contact( #CYL.FULL_CLOSED )
      Coil( #HMI_MOTION_END_POS_RIGHT )
   END_RUNG
   RUNG wire#w1
      Contact( #PRESSURE_RELEASED )
      Coil( #HMI_MOTION_END_POS_LEFT_2 )
   END_RUNG
   RUNG wire#w1
      Contact( #CYL.FULL_LOW_PRESSURED )
      Coil( #HMI_MOTION_END_POS_RIGHT_2 )
   END_RUNG
   // the same network as SCL:
   #HMI_MOTION_END_POS_LEFT := "M_ONE" AND #CYL.FULL_OPEN;
   #HMI_MOTION_END_POS_RIGHT := "M_ONE" AND #CYL.FULL_CLOSED;
   #HMI_MOTION_END_POS_LEFT_2 := "M_ONE" AND #PRESSURE_RELEASED;
   #HMI_MOTION_END_POS_RIGHT_2 := "M_ONE" AND #CYL.FULL_LOW_PRESSURED;
END_REGION

REGION Network 110: HMI STATUS
   RUNG wire#powerrail
      Contact( "M_0.5_SEC_2HZ" )
      wire#w1
      Contact( #OPEN_ACTION )
      I_Contact( #OPEN_STATUS )
      Coil( #HMI_MOTION_ACTIVE_LEFT )
   END_RUNG
   RUNG wire#w1
      Contact( #CLOSE )
      I_Contact( #CLOSED )
      Coil( #HMI_MOTION_ACTIVE_RIGHT )
   END_RUNG
   RUNG wire#w1
      Contact( #CYL.RELEASE_PRESSURE_COMMAND )
      I_Contact( #PRESSURE_RELEASED )
      Coil( #HMI_MOTION_ACTIVE_LEFT_2 )
   END_RUNG
   RUNG wire#w1
      Contact( #LOW_PRESSURE )
      I_Contact( #LOW_PRESSURED )
      Coil( #HMI_MOTION_ACTIVE_RIGHT_2 )
   END_RUNG
   // the same network as SCL:
   #HMI_MOTION_ACTIVE_LEFT := "M_0.5_SEC_2HZ" AND #OPEN_ACTION AND NOT #OPEN_STATUS;
   #HMI_MOTION_ACTIVE_RIGHT := "M_0.5_SEC_2HZ" AND #CLOSE AND NOT #CLOSED;
   #HMI_MOTION_ACTIVE_LEFT_2 := "M_0.5_SEC_2HZ" AND #CYL.RELEASE_PRESSURE_COMMAND AND NOT #PRESSURE_RELEASED;
   #HMI_MOTION_ACTIVE_RIGHT_2 := "M_0.5_SEC_2HZ" AND #LOW_PRESSURE AND NOT #LOW_PRESSURED;
END_REGION

REGION Network 111: HMI FLOWMETER SCREEN CLOSED LOW AUXILIARY
   RUNG wire#powerrail
      Contact( #LOW_PRESSURED )
      Contact( #CYL.CLOSE_LOW_PRESSURE )
      Coil( #CYL.HMI_ACTD_LOW_AUX )
   END_RUNG
   // the same network as SCL:
   #CYL.HMI_ACTD_LOW_AUX := #LOW_PRESSURED AND #CYL.CLOSE_LOW_PRESSURE;
END_REGION

REGION Network 112: HMI FLOWMETER SCREEN OPEN LOW AUXILIARY
   RUNG wire#powerrail
      Contact( #LOW_PRESSURED )
      Contact( #CYL.OPEN_LOW_PRESSURE )
      Coil( #CYL.HMI_DEACTD_LOW_AUX )
   END_RUNG
   // the same network as SCL:
   #CYL.HMI_DEACTD_LOW_AUX := #LOW_PRESSURED AND #CYL.OPEN_LOW_PRESSURE;
END_REGION

REGION Network 113: RESET FLOWMETER
   RUNG wire#powerrail
      Contact( #OPEN_STATUS )
      P_Trig( #CYL.PULSE_1 )
      Contact( #OPEN_ACTION )
      wire#w1
      Coil( #RESET_FLOWMETER )
   END_RUNG
   RUNG wire#powerrail
      Contact( #OPEN_STATUS )
      N_Trig( #CYL.PULSE_2 )
      Contact( #CLOSE )
   END_RUNG wire#w1
   RUNG wire#powerrail
      Contact( #OPEN_ACTION )
      Contact( #CYL.TIME_EXCEEDED_ALARM )
      P_Trig( #CYL.PULSE_3 )
      Contact( #OPEN_FLOW_ACTIVE_FLOWMETER )
   END_RUNG wire#w1
   RUNG wire#powerrail
      Contact( #FLOWMETER_RESET )
      P_Trig( #CYL.PULSE_4 )
   END_RUNG wire#w1
   RUNG wire#powerrail
      Contact( "M_FIRST_SCAN" )
   END_RUNG wire#w1
   RUNG wire#w1
      R_Coil( #OPEN_FLOW_ACTIVE_FLOWMETER )
   END_RUNG
   // the same network as SCL:
   #_w1 := #OPEN_STATUS AND NOT #CYL.PULSE_1;   // rising edge
   #CYL.PULSE_1 := #OPEN_STATUS;
   #_w2 := NOT #OPEN_STATUS AND #CYL.PULSE_2;   // falling edge
   #CYL.PULSE_2 := #OPEN_STATUS;
   #_w3 := #OPEN_ACTION AND #CYL.TIME_EXCEEDED_ALARM;
   #_w4 := #_w3 AND NOT #CYL.PULSE_3;   // rising edge
   #CYL.PULSE_3 := #_w3;
   #_w5 := #FLOWMETER_RESET AND NOT #CYL.PULSE_4;   // rising edge
   #CYL.PULSE_4 := #FLOWMETER_RESET;
   #RESET_FLOWMETER := (#_w1 AND #OPEN_ACTION) OR (#_w2 AND #CLOSE) OR (#_w4 AND #OPEN_FLOW_ACTIVE_FLOWMETER) OR #_w5 OR "M_FIRST_SCAN";
   IF #RESET_FLOWMETER THEN #OPEN_FLOW_ACTIVE_FLOWMETER := FALSE; END_IF;
END_REGION
END_FUNCTION_BLOCK
